(* IEC 61131-3 sources: verifaps-lib/symbex/src/test/resources/edu/kit/iti/formal/automation/st/stoo/integration, 2 files *)

(* ---- effective_subtypes.st ---- *)
INTERFACE ITF
  METHOD f : INT
    VAR_INPUT
      x : INT;
    END_VAR
  END_METHOD
END_INTERFACE

CLASS A IMPLEMENTS ITF
  VAR
    b1 : B;
    b2 : B;
    c1 : C;
    c2 : C;
  END_VAR

  METHOD f : INT
    VAR_INPUT
      x : INT;
    END_VAR

    f := 42;
  END_METHOD
END_CLASS

CLASS A1 EXTENDS A
  METHOD f : INT
    VAR_INPUT
      x : INT;
    END_VAR

    f := 24;
  END_METHOD
END_CLASS

CLASS A2 EXTENDS A
  METHOD f : INT
    VAR_INPUT
      x : INT;
    END_VAR

    f := 33;
  END_METHOD
END_CLASS

CLASS B IMPLEMENTS ITF
  VAR
    c1 : C;
    c2 : C;
  END_VAR
END_CLASS

CLASS C
END_CLASS

PROGRAM MY_PROGRAM
  VAR_INPUT
    switch : BOOL;
    x : INT;
  END_VAR
  VAR
    i : ITF;
    a : A;
    a1 : A1;
    b : B;
    r : REF_TO A;
  END_VAR
  VAR_OUTPUT
    y : INT;
  END_VAR

  r := REF(a1);

  IF (switch) THEN
    i := a;
  ELSE
    i := b;
  END_IF

  y := r^.f(x);

  r^.c1 := a.b1.c1;
  r^.c2 := a.b2.c2;

  r^.b1.c2 := r^.c2;
END_PROGRAM

(* ---- simple_hierarchy.st ---- *)
CLASS A
  VAR
    x : INT;
    y : INT;
  END_VAR

  METHOD f : INT
    f := x + y;
  END_METHOD

  METHOD g : INT
    g := x * y;
  END_METHOD
END_CLASS

CLASS B EXTENDS A
  VAR
    z : INT;
  END_VAR

  METHOD OVERRIDE f : INT
    f := SUPER.f() + z;
  END_METHOD

  METHOD OVERRIDE g : INT
    g := x * y * z;
  END_METHOD
END_CLASS

CLASS C EXTENDS B
  VAR
    r : INT;
  END_VAR

  METHOD OVERRIDE g : INT
    g := r * x * y * z;
  END_METHOD
END_CLASS

PROGRAM MY_PROGRAM
  VAR
    a : A := (x := 42, y := 24);
    b : B := (x := 33, y := 44, z := 55);
    c : C := (x := 1, y := 2, z := 3, r := 4);
  END_VAR
  VAR_OUTPUT
    x : INT;
    y : INT;
  END_VAR

  y := c.f();
  x := c.x;
END_PROGRAM
